PROGRAM MAIN
VAR
	disposable_TestSuite : Disposable_TestSuite;
END_VAR

TcUnit.RUN();

END_PROGRAM

(* stored: Version 1.1.0.1, ProductVersion 3.1.4024.12
   POU MAIN: Id {9d67fa5f-b22b-413d-bd2f-078ef7b27582}, SpecialFunc None *)
